{attribute 'GeneratedUsingTerminal: EL2262-0000-0001'}
{attribute addProperty BoxType "EL2262-0000-0001"}
{attribute addProperty Id "EtcSlaveTerminalBaseCycCount0AT %Q*CycCount0_2C2338042Sample0_0AT %Q*Sample_0023574C1GapAT %I*EMPTY_STRUCTURE0CycCount1AT %Q*CycCount1_2C2338042Sample1_0AT %Q*Sample_07D5B44A1Gap_1AT %I*EMPTY_STRUCTURE0WcStateAT %I*WcState_0B2B16F91InfoDataAT %I*InfoData_A7436BC610"}
{attribute addProperty CRC "1442097891"}
{attribute addProperty Size "17"}
TYPE EL2262_55F4AAE3 EXTENDS EtcSlaveTerminalBase :
STRUCT
	{attribute addProperty Name "CycCount0"}
	CycCount0 : CycCount0_2C233804;
	{attribute addProperty Name "Sample0_0"}
	Sample0_0 : Sample_0023574C;
	{attribute addProperty Name "Gap"}
	Gap : EMPTY_STRUCTURE;
	{attribute addProperty Name "CycCount1"}
	CycCount1 : CycCount1_2C233804;
	{attribute addProperty Name "Sample1_0"}
	Sample1_0 : Sample_07D5B44A;
	{attribute addProperty Name "Gap_1"}
	Gap_1 : EMPTY_STRUCTURE;
	{attribute addProperty Name "WcState"}
	WcState : WcState_0B2B16F9;
	{attribute addProperty Name "InfoData"}
	InfoData : InfoData_A7436BC6;
END_STRUCT
END_TYPE

(* stored: Version 1.2.0.0, ProductVersion 3.1.4024.9
   DUT EL2262_55F4AAE3: Id {8ca43887-92fa-416e-816e-959a7125d715} *)
